TYPE ST_AteqBitmapReadErrorCode :
STRUCT
END_STRUCT
END_TYPE

(* stored: Version 1.1.0.1, ProductVersion 3.1.4024.15
   DUT ST_AteqBitmapReadErrorCode: Id {2bf05f50-b411-4198-ab9d-a432a2ca1a9f} *)
